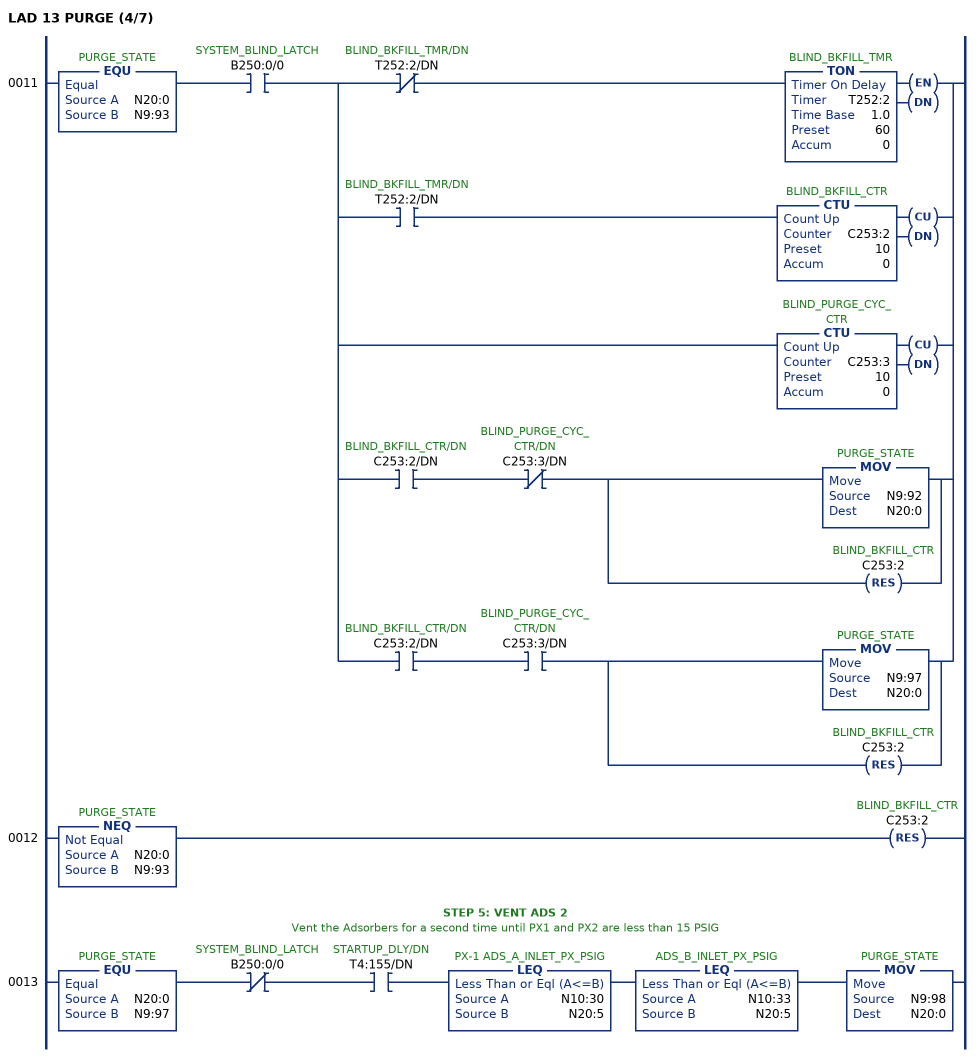
% Rung: 11 %
SOR EQU N20:0 N9:93 XIC B250:0/0 BST XIO T252:2/DN TON T252:2 1.0 60 0 NXB XIC T252:2/DN CTU C253:2 10 0 NXB CTU C253:3 10 0 NXB XIC C253:2/DN XIO C253:3/DN BST MOV N9:92 N20:0 NXB RES C253:2 BND NXB XIC C253:2/DN XIC C253:3/DN BST MOV N9:97 N20:0 NXB RES C253:2 BND BND EOR
%   N20:0  PURGE_STATE %
%   N9:93  PURGE_BACKFILL %
%   B250:0/0  SYSTEM_BLIND_LATCH %
%   T252:2  BLIND_BKFILL_TMR %
%   C253:2  BLIND_BKFILL_CTR %
%   C253:3  BLIND_PURGE_CYC_CTR %
%   N9:92  PURGE_VENT_ADSORBER %
%   N9:97  PURGE_VENT_ADS_2 %
% Rung: 12 %
SOR NEQ N20:0 N9:93 RES C253:2 EOR
%   N20:0  PURGE_STATE %
%   N9:93  PURGE_BACKFILL %
%   C253:2  BLIND_BKFILL_CTR %
% Rung: 13 %
% TITLE: STEP 5: VENT ADS 2 %
% Vent the Adsorbers for a second time until PX1 and PX2 are less than 15 PSIG %
SOR EQU N20:0 N9:97 XIO B250:0/0 XIC T4:155/DN LEQ N10:30 N20:5 LEQ N10:33 N20:5 MOV N9:98 N20:0 EOR
%   N20:0  PURGE_STATE %
%   N9:97  PURGE_VENT_ADS_2 %
%   B250:0/0  SYSTEM_BLIND_LATCH %
%   T4:155  STARTUP_DLY %
%   N10:30  ADS_A_INLET_PX_PSIG  "PX-1" %
%   N20:5  PURGE_VENT_ADS_2_PX %
%   N10:33  ADS_B_INLET_PX_PSIG %
%   N9:98  PURGE_VENT_GET_2 %

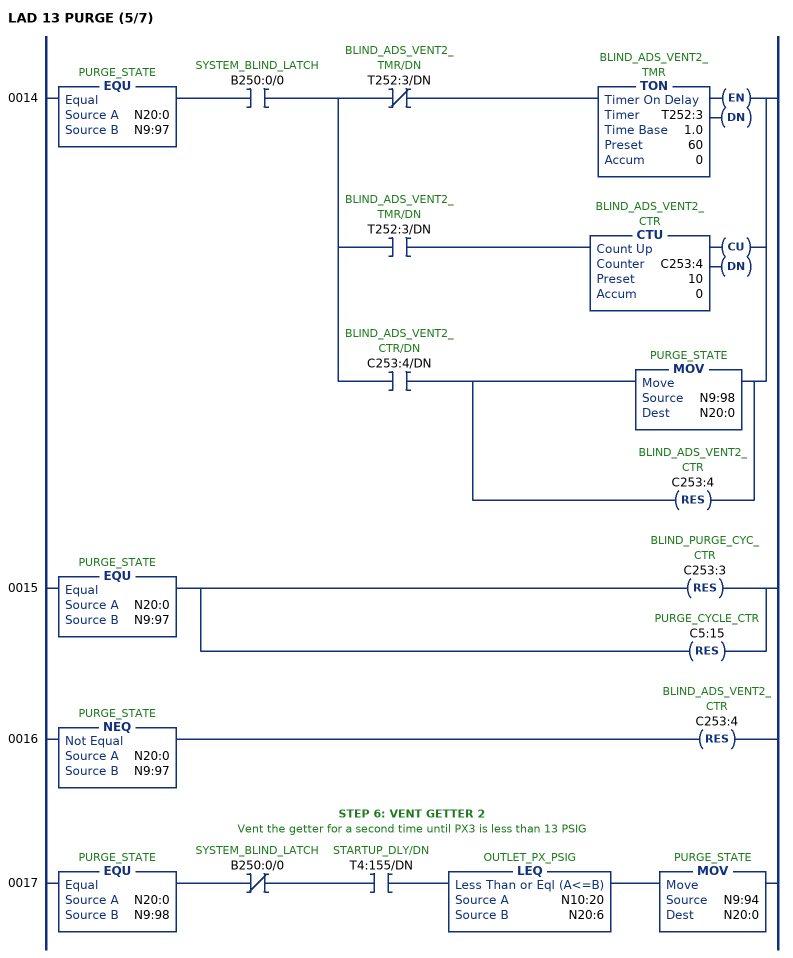
% Rung: 14 %
SOR EQU N20:0 N9:97 XIC B250:0/0 BST XIO T252:3/DN TON T252:3 1.0 60 0 NXB XIC T252:3/DN CTU C253:4 10 0 NXB XIC C253:4/DN BST MOV N9:98 N20:0 NXB RES C253:4 BND BND EOR
%   N20:0  PURGE_STATE %
%   N9:97  PURGE_VENT_ADS_2 %
%   B250:0/0  SYSTEM_BLIND_LATCH %
%   T252:3  BLIND_ADS_VENT2_TMR %
%   C253:4  BLIND_ADS_VENT2_CTR %
%   N9:98  PURGE_VENT_GET_2 %
% Rung: 15 %
SOR EQU N20:0 N9:97 BST RES C253:3 NXB RES C5:15 BND EOR
%   N20:0  PURGE_STATE %
%   N9:97  PURGE_VENT_ADS_2 %
%   C253:3  BLIND_PURGE_CYC_CTR %
%   C5:15  PURGE_CYCLE_CTR %
% Rung: 16 %
SOR NEQ N20:0 N9:97 RES C253:4 EOR
%   N20:0  PURGE_STATE %
%   N9:97  PURGE_VENT_ADS_2 %
%   C253:4  BLIND_ADS_VENT2_CTR %
% Rung: 17 %
% TITLE: STEP 6: VENT GETTER 2 %
% Vent the getter for a second time until PX3 is less than 13 PSIG %
SOR EQU N20:0 N9:98 XIO B250:0/0 XIC T4:155/DN LEQ N10:20 N20:6 MOV N9:94 N20:0 EOR
%   N20:0  PURGE_STATE %
%   N9:98  PURGE_VENT_GET_2 %
%   B250:0/0  SYSTEM_BLIND_LATCH %
%   T4:155  STARTUP_DLY %
%   N10:20  OUTLET_PX_PSIG %
%   N20:6  PURGE_VENT_GET_2_PX %
%   N9:94  PURGE_FINAL_VENT %

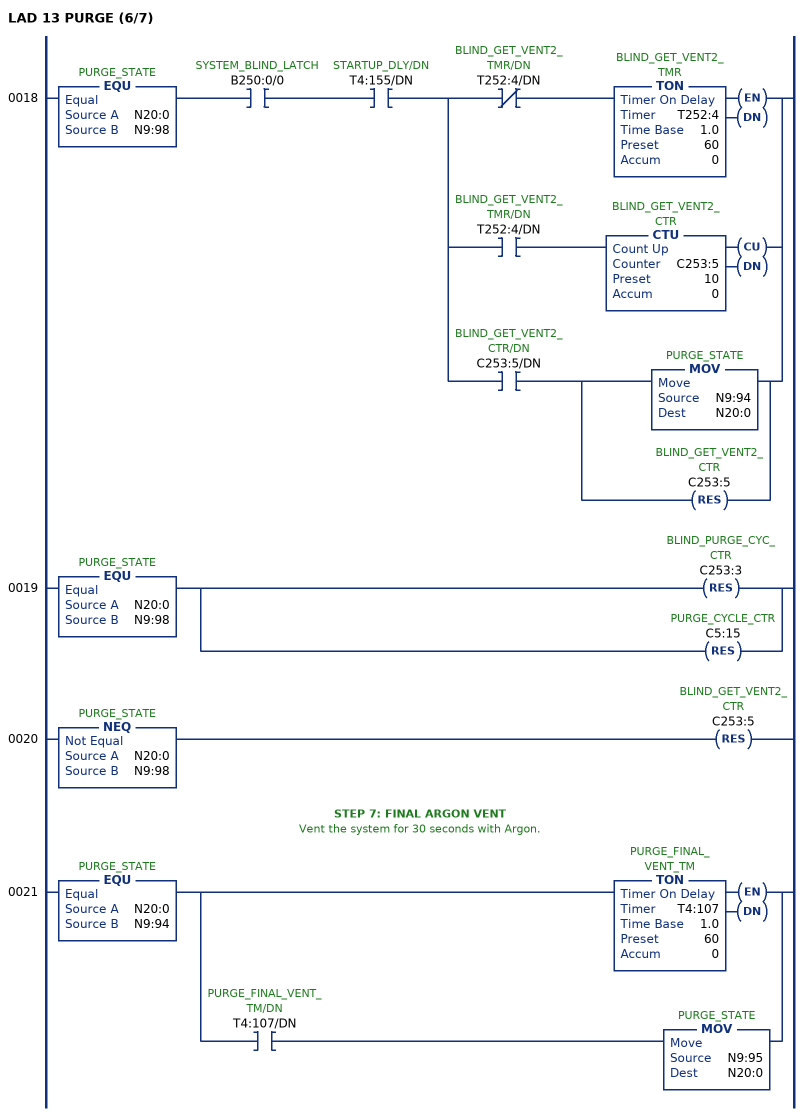
% Rung: 18 %
SOR EQU N20:0 N9:98 XIC B250:0/0 XIC T4:155/DN BST XIO T252:4/DN TON T252:4 1.0 60 0 NXB XIC T252:4/DN CTU C253:5 10 0 NXB XIC C253:5/DN BST MOV N9:94 N20:0 NXB RES C253:5 BND BND EOR
%   N20:0  PURGE_STATE %
%   N9:98  PURGE_VENT_GET_2 %
%   B250:0/0  SYSTEM_BLIND_LATCH %
%   T4:155  STARTUP_DLY %
%   T252:4  BLIND_GET_VENT2_TMR %
%   C253:5  BLIND_GET_VENT2_CTR %
%   N9:94  PURGE_FINAL_VENT %
% Rung: 19 %
SOR EQU N20:0 N9:98 BST RES C253:3 NXB RES C5:15 BND EOR
%   N20:0  PURGE_STATE %
%   N9:98  PURGE_VENT_GET_2 %
%   C253:3  BLIND_PURGE_CYC_CTR %
%   C5:15  PURGE_CYCLE_CTR %
% Rung: 20 %
SOR NEQ N20:0 N9:98 RES C253:5 EOR
%   N20:0  PURGE_STATE %
%   N9:98  PURGE_VENT_GET_2 %
%   C253:5  BLIND_GET_VENT2_CTR %
% Rung: 21 %
% TITLE: STEP 7: FINAL ARGON VENT %
% Vent the system for 30 seconds with Argon. %
SOR EQU N20:0 N9:94 BST TON T4:107 1.0 60 0 NXB XIC T4:107/DN MOV N9:95 N20:0 BND EOR
%   N20:0  PURGE_STATE %
%   N9:94  PURGE_FINAL_VENT %
%   T4:107  PURGE_FINAL_VENT_TM %
%   N9:95  PURGE_DONE %

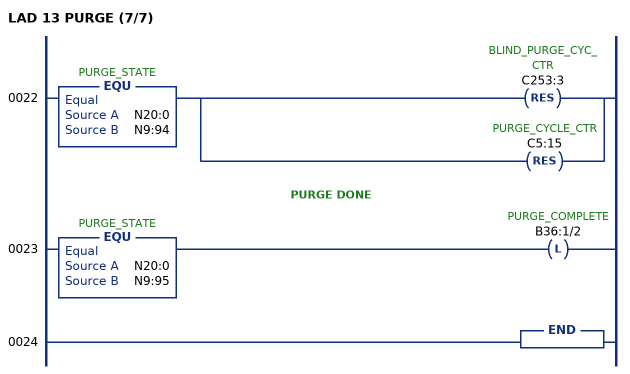
% Rung: 22 %
SOR EQU N20:0 N9:94 BST RES C253:3 NXB RES C5:15 BND EOR
%   N20:0  PURGE_STATE %
%   N9:94  PURGE_FINAL_VENT %
%   C253:3  BLIND_PURGE_CYC_CTR %
%   C5:15  PURGE_CYCLE_CTR %
% Rung: 23 %
% TITLE: PURGE DONE %
SOR EQU N20:0 N9:95 OTL B36:1/2 EOR
%   N20:0  PURGE_STATE %
%   N9:95  PURGE_DONE %
%   B36:1/2  PURGE_COMPLETE %
% Rung: 24 %
SOR END EOR

LADDER 14 "MFM"
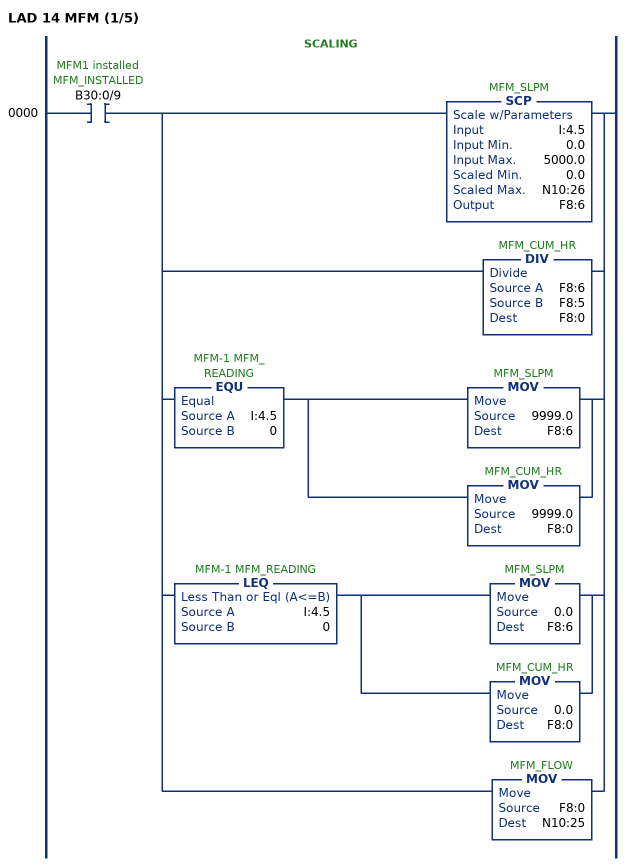
% Rung: 0 %
% TITLE: SCALING %
SOR XIC B30:0/9 BST SCP I:4.5 0.0 5000.0 0.0 N10:26 F8:6 NXB DIV F8:6 F8:5 F8:0 NXB EQU I:4.5 0 BST MOV 9999.0 F8:6 NXB MOV 9999.0 F8:0 BND NXB LEQ I:4.5 0 BST MOV 0.0 F8:6 NXB MOV 0.0 F8:0 BND NXB MOV F8:0 N10:25 BND EOR
%   B30:0/9  MFM_INSTALLED  "MFM1 installed" %
%   I:4.5  MFM_READING  "MFM-1" %
%   N10:26  MFM_SCALING %
%   F8:6  MFM_SLPM %
%   F8:5  CUM_TO_SLPM %
%   F8:0  MFM_CUM_HR %
%   N10:25  MFM_FLOW %

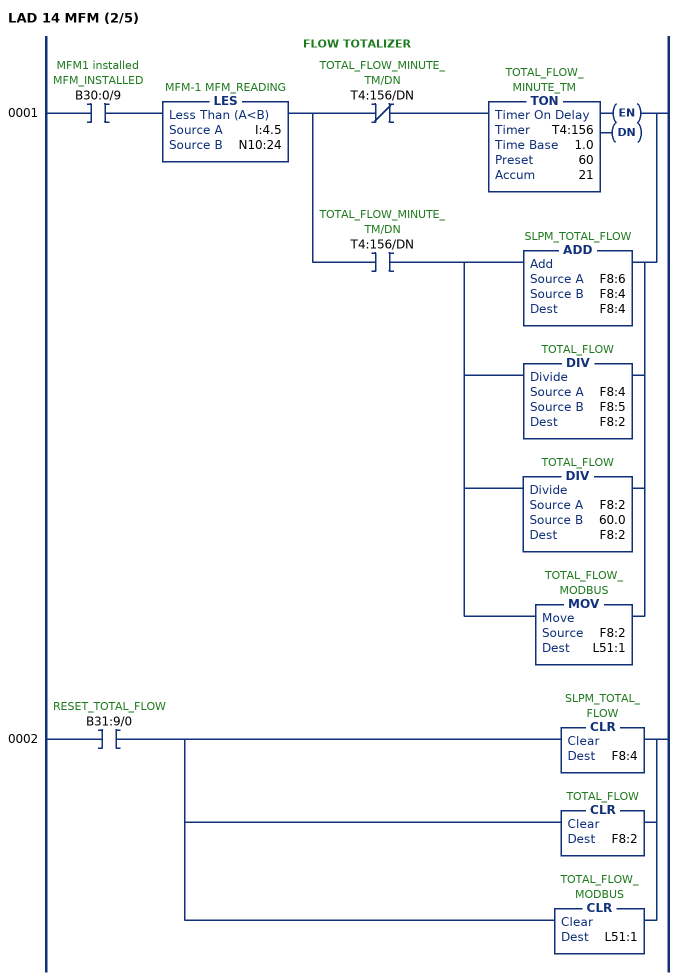
% Rung: 1 %
% TITLE: FLOW TOTALIZER %
SOR XIC B30:0/9 LES I:4.5 N10:24 BST XIO T4:156/DN TON T4:156 1.0 60 21 NXB XIC T4:156/DN BST ADD F8:6 F8:4 F8:4 NXB DIV F8:4 F8:5 F8:2 NXB DIV F8:2 60.0 F8:2 NXB MOV F8:2 L51:1 BND BND EOR
%   B30:0/9  MFM_INSTALLED  "MFM1 installed" %
%   I:4.5  MFM_READING  "MFM-1" %
%   N10:24  OPEN_MFM_5V %
%   T4:156  TOTAL_FLOW_MINUTE_TM %
%   F8:6  MFM_SLPM %
%   F8:4  SLPM_TOTAL_FLOW %
%   F8:5  CUM_TO_SLPM %
%   F8:2  TOTAL_FLOW %
%   L51:1  TOTAL_FLOW_MODBUS %
% Rung: 2 %
SOR XIC B31:9/0 BST CLR F8:4 NXB CLR F8:2 NXB CLR L51:1 BND EOR
%   B31:9/0  RESET_TOTAL_FLOW %
%   F8:4  SLPM_TOTAL_FLOW %
%   F8:2  TOTAL_FLOW %
%   L51:1  TOTAL_FLOW_MODBUS %

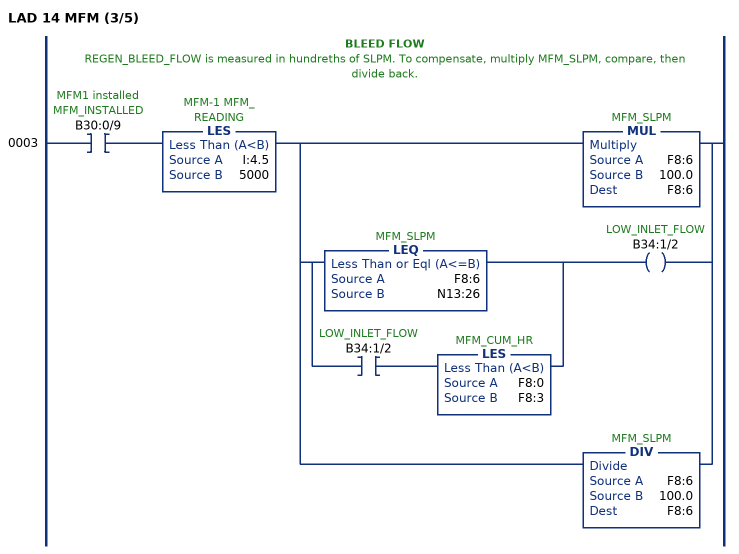
% Rung: 3 %
% TITLE: BLEED FLOW %
% REGEN_BLEED_FLOW is measured in hundreths of SLPM. To compensate, multiply MFM_SLPM, compare, then divide back. %
SOR XIC B30:0/9 LES I:4.5 5000 BST MUL F8:6 100.0 F8:6 NXB BST LEQ F8:6 N13:26 NXB XIC B34:1/2 LES F8:0 F8:3 BND OTE B34:1/2 NXB DIV F8:6 100.0 F8:6 BND EOR
%   B30:0/9  MFM_INSTALLED  "MFM1 installed" %
%   I:4.5  MFM_READING  "MFM-1" %
%   F8:6  MFM_SLPM %
%   N13:26  REGEN_BLEED_FLOW %
%   B34:1/2  LOW_INLET_FLOW %
%   F8:0  MFM_CUM_HR %
%   F8:3  BLEED_FLOW_CUTOFF %

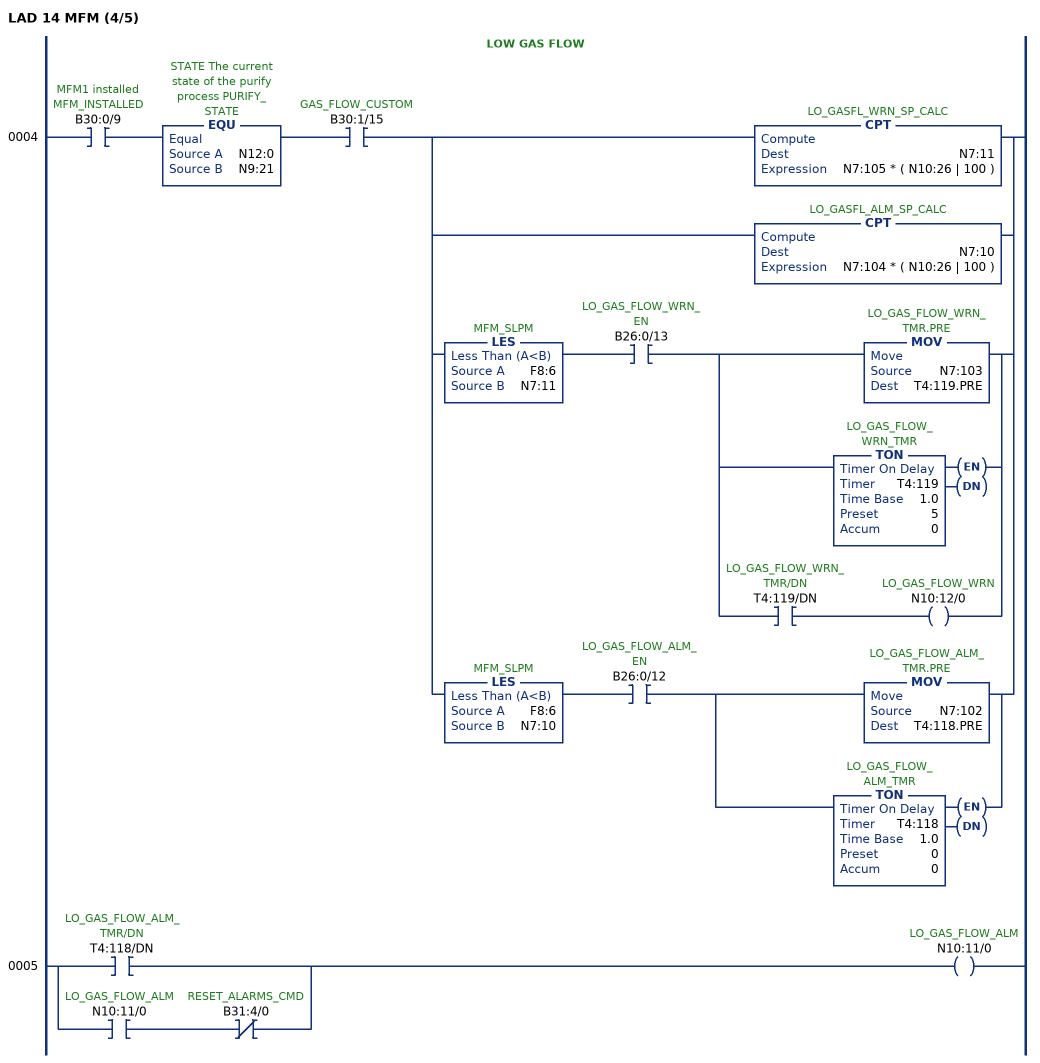
% Rung: 4 %
% TITLE: LOW GAS FLOW %
SOR XIC B30:0/9 EQU N12:0 N9:21 XIC B30:1/15 BST CPT N7:11 " N7:105 * ( N10:26 | 100 ) " NXB CPT N7:10 " N7:104 * ( N10:26 | 100 ) " NXB LES F8:6 N7:11 XIC B26:0/13 BST MOV N7:103 T4:119.PRE NXB TON T4:119 1.0 5 0 NXB XIC T4:119/DN OTE N10:12/0 BND NXB LES F8:6 N7:10 XIC B26:0/12 BST MOV N7:102 T4:118.PRE NXB TON T4:118 1.0 0 0 BND BND EOR
%   B30:0/9  MFM_INSTALLED  "MFM1 installed" %
%   N12:0  PURIFY_STATE  "STATE The current state of the purify process" %
%   N9:21  PURIFY_RUN  "STATE Purify running" %
%   B30:1/15  GAS_FLOW_CUSTOM %
%   N7:11  LO_GASFL_WRN_SP_CALC %
%   N7:105  LO_GAS_FLOW_WRN_SP %
%   N10:26  MFM_SCALING %
%   N7:10  LO_GASFL_ALM_SP_CALC %
%   N7:104  LO_GAS_FLOW_ALM_SP %
%   F8:6  MFM_SLPM %
%   B26:0/13  LO_GAS_FLOW_WRN_EN %
%   N7:103  LO_GAS_FLOW_WRN_DLY %
%   T4:119  LO_GAS_FLOW_WRN_TMR %
%   N10:12/0  LO_GAS_FLOW_WRN %
%   B26:0/12  LO_GAS_FLOW_ALM_EN %
%   N7:102  LO_GAS_FLOW_ALM_DLY %
%   T4:118  LO_GAS_FLOW_ALM_TMR %
% Rung: 5 %
SOR BST XIC T4:118/DN NXB XIC N10:11/0 XIO B31:4/0 BND OTE N10:11/0 EOR
%   T4:118  LO_GAS_FLOW_ALM_TMR %
%   N10:11/0  LO_GAS_FLOW_ALM %
%   B31:4/0  RESET_ALARMS_CMD %

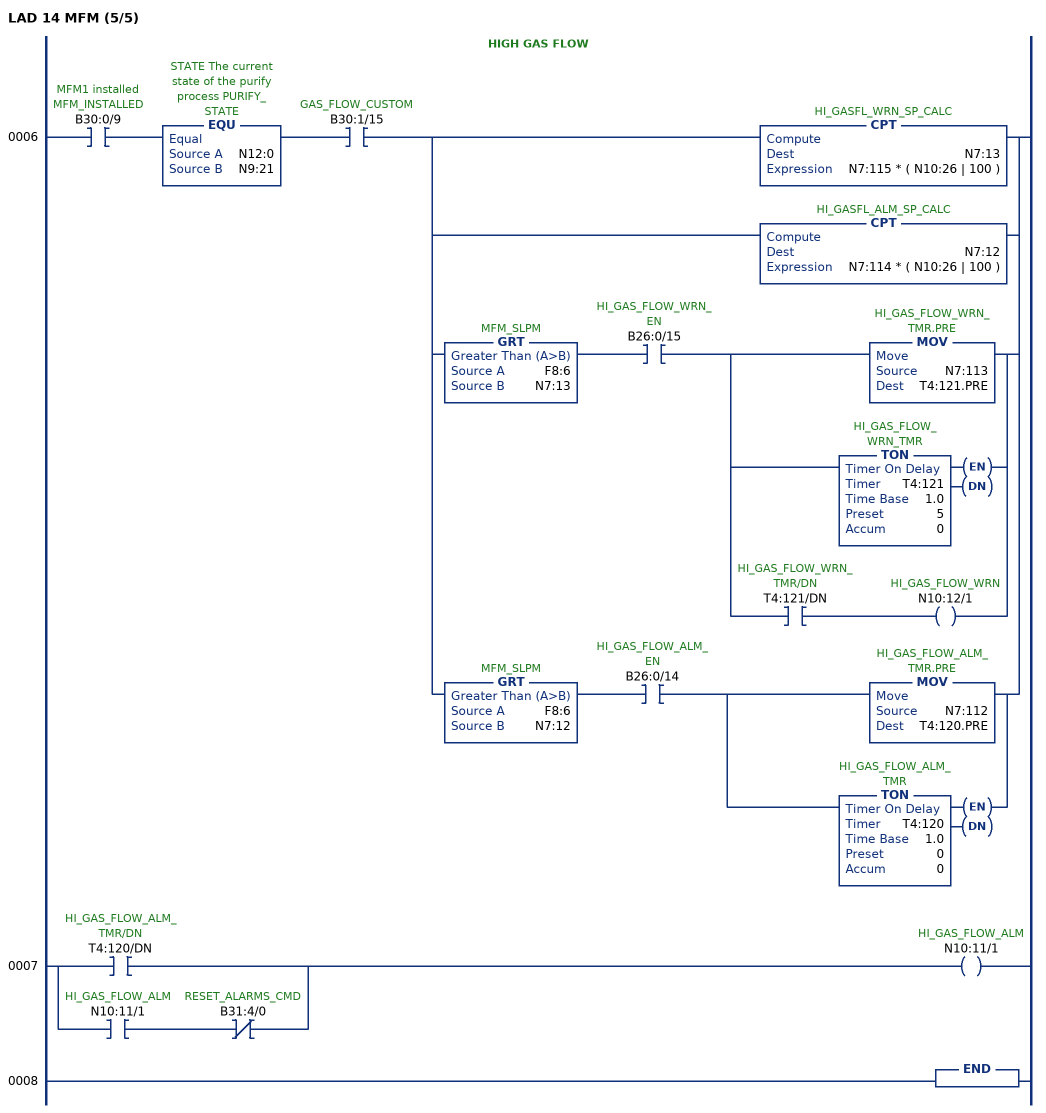
% Rung: 6 %
% TITLE: HIGH GAS FLOW %
SOR XIC B30:0/9 EQU N12:0 N9:21 XIC B30:1/15 BST CPT N7:13 " N7:115 * ( N10:26 | 100 ) " NXB CPT N7:12 " N7:114 * ( N10:26 | 100 ) " NXB GRT F8:6 N7:13 XIC B26:0/15 BST MOV N7:113 T4:121.PRE NXB TON T4:121 1.0 5 0 NXB XIC T4:121/DN OTE N10:12/1 BND NXB GRT F8:6 N7:12 XIC B26:0/14 BST MOV N7:112 T4:120.PRE NXB TON T4:120 1.0 0 0 BND BND EOR
%   B30:0/9  MFM_INSTALLED  "MFM1 installed" %
%   N12:0  PURIFY_STATE  "STATE The current state of the purify process" %
%   N9:21  PURIFY_RUN  "STATE Purify running" %
%   B30:1/15  GAS_FLOW_CUSTOM %
%   N7:13  HI_GASFL_WRN_SP_CALC %
%   N7:115  HI_GAS_FLOW_WRN_SP %
%   N10:26  MFM_SCALING %
%   N7:12  HI_GASFL_ALM_SP_CALC %
%   N7:114  HI_GAS_FLOW_ALM_SP %
%   F8:6  MFM_SLPM %
%   B26:0/15  HI_GAS_FLOW_WRN_EN %
%   N7:113  HI_GAS_FLOW_WRN_DLY %
%   T4:121  HI_GAS_FLOW_WRN_TMR %
%   N10:12/1  HI_GAS_FLOW_WRN %
%   B26:0/14  HI_GAS_FLOW_ALM_EN %
%   N7:112  HI_GAS_FLOW_ALM_DLY %
%   T4:120  HI_GAS_FLOW_ALM_TMR %
% Rung: 7 %
SOR BST XIC T4:120/DN NXB XIC N10:11/1 XIO B31:4/0 BND OTE N10:11/1 EOR
%   T4:120  HI_GAS_FLOW_ALM_TMR %
%   N10:11/1  HI_GAS_FLOW_ALM %
%   B31:4/0  RESET_ALARMS_CMD %
% Rung: 8 %
SOR END EOR

LADDER 16 "MFC"
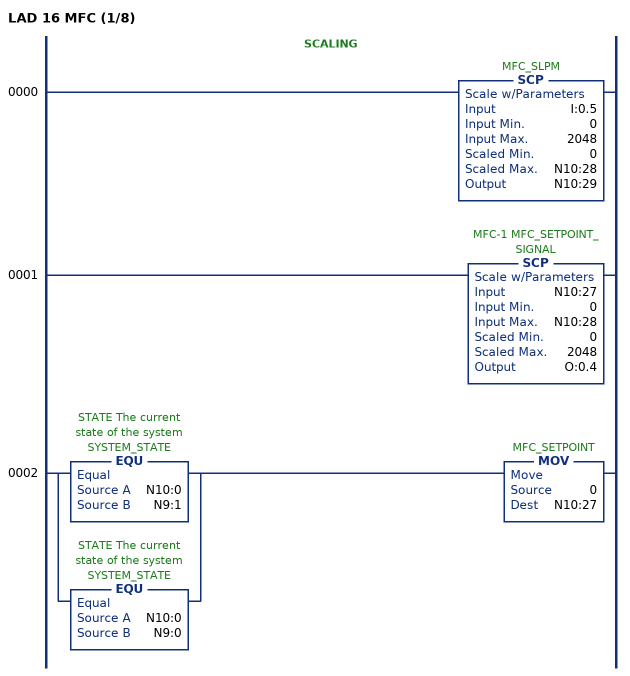
% Rung: 0 %
% TITLE: SCALING %
SOR SCP I:0.5 0 2048 0 N10:28 N10:29 EOR
%   I:0.5  MFC_FEEDBACK  "MFC-1" %
%   N10:28  MFC_SCALING  "in slpm" %
%   N10:29  MFC_SLPM %
% Rung: 1 %
SOR SCP N10:27 0 N10:28 0 2048 O:0.4 EOR
%   N10:27  MFC_SETPOINT %
%   N10:28  MFC_SCALING  "in slpm" %
%   O:0.4  MFC_SETPOINT_SIGNAL  "MFC-1" %
% Rung: 2 %
SOR BST EQU N10:0 N9:1 NXB EQU N10:0 N9:0 BND MOV 0 N10:27 EOR
%   N10:0  SYSTEM_STATE  "STATE The current state of the system" %
%   N9:1  SYSTEM_STANDBY  "STATE System Process" %
%   N9:0  SYSTEM_OFFLINE %
%   N10:27  MFC_SETPOINT %

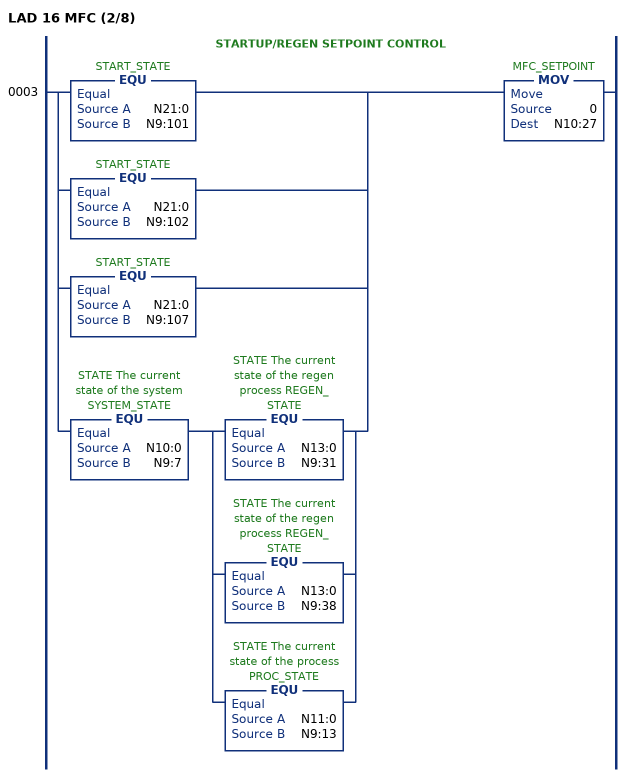
% Rung: 3 %
% TITLE: STARTUP/REGEN SETPOINT CONTROL %
SOR BST EQU N21:0 N9:101 NXB EQU N21:0 N9:102 NXB EQU N21:0 N9:107 NXB EQU N10:0 N9:7 BST EQU N13:0 N9:31 NXB EQU N13:0 N9:38 NXB EQU N11:0 N9:13 BND BND MOV 0 N10:27 EOR
%   N21:0  START_STATE %
%   N9:101  START_COOL %
%   N9:102  START_VENT_ADS_1 %
%   N9:107  START_VENT_ADS_2 %
%   N10:0  SYSTEM_STATE  "STATE The current state of the system" %
%   N9:7  SYSTEM_COLD_START %
%   N13:0  REGEN_STATE  "STATE The current state of the regen process" %
%   N9:31  REGEN_DELAY  "STATE Regen Delay" %
%   N9:38  REGEN_DONE %
%   N11:0  PROC_STATE  "STATE The current state of the process" %
%   N9:13  PROC_OVERLAP  "STATE Process Purify Overlap" %
%   N10:27  MFC_SETPOINT %

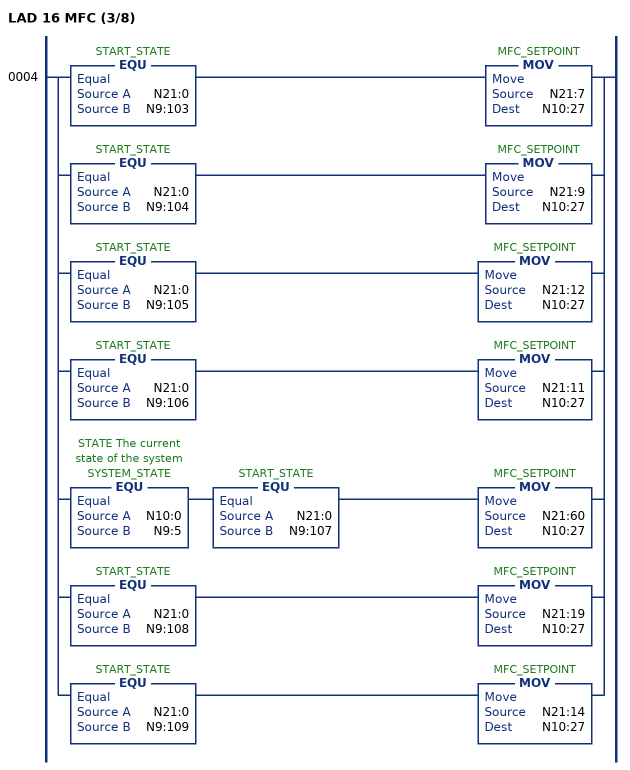
% Rung: 4 %
SOR BST EQU N21:0 N9:103 MOV N21:7 N10:27 NXB EQU N21:0 N9:104 MOV N21:9 N10:27 NXB EQU N21:0 N9:105 MOV N21:12 N10:27 NXB EQU N21:0 N9:106 MOV N21:11 N10:27 NXB EQU N10:0 N9:5 EQU N21:0 N9:107 MOV N21:60 N10:27 NXB EQU N21:0 N9:108 MOV N21:19 N10:27 NXB EQU N21:0 N9:109 MOV N21:14 N10:27 BND EOR
%   N21:0  START_STATE %
%   N9:103  START_VENT_GET_1 %
%   N21:7  START_VENT_GET_1_FLW %
%   N10:27  MFC_SETPOINT %
%   N9:104  START_HEAT_GETTER %
%   N21:9  START_HEAT_FLW %
%   N9:105  START_VENT_ALL %
%   N21:12  START_VENT_ALL_FLW %
%   N9:106  START_BACKFILL_1 %
%   N21:11  START_BKFIL_1_FLW %
%   N10:0  SYSTEM_STATE  "STATE The current state of the system" %
%   N9:5  SYSTEM_QUICK_START %
%   N9:107  START_VENT_ADS_2 %
%   N21:60  START_VENT_ADS_2_FLW %
%   N9:108  START_VENT_GET_2 %
%   N21:19  START_VENT_GET_2_FLW %
%   N9:109  START_BKFL_2 %
%   N21:14  START_BKFIL_2_FLW %

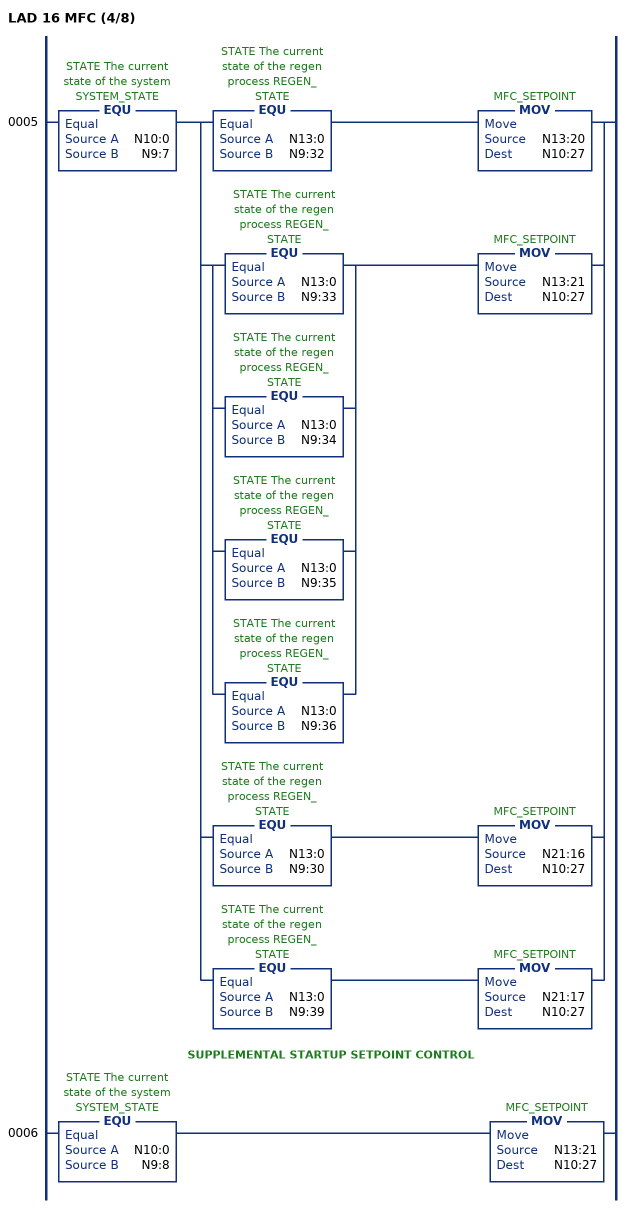
% Rung: 5 %
SOR EQU N10:0 N9:7 BST EQU N13:0 N9:32 MOV N13:20 N10:27 NXB BST EQU N13:0 N9:33 NXB EQU N13:0 N9:34 NXB EQU N13:0 N9:35 NXB EQU N13:0 N9:36 BND MOV N13:21 N10:27 NXB EQU N13:0 N9:30 MOV N21:16 N10:27 NXB EQU N13:0 N9:39 MOV N21:17 N10:27 BND EOR
%   N10:0  SYSTEM_STATE  "STATE The current state of the system" %
%   N9:7  SYSTEM_COLD_START %
%   N13:0  REGEN_STATE  "STATE The current state of the regen process" %
%   N9:32  REGEN_VENT  "STATE Regen Vent" %
%   N13:20  REGEN_VENT_FLOW %
%   N10:27  MFC_SETPOINT %
%   N9:33  REGEN_HEAT_BED  "STATE Regen Heat wall" %
%   N9:34  REGEN_RUN  "STATE Regen Running" %
%   N9:35  REGEN_COOL_WALL  "STATE Regen Cool wall" %
%   N9:36  REGEN_COOL  "STATE Regen Cool" %
%   N13:21  REGEN_MAIN_FLOW %
%   N9:30  REGEN_STANDBY  "STATE Regen Standby" %
%   N21:16  START_REG_BLEED_FLW %
%   N9:39  REGEN_BACKFILL %
%   N21:17  START_REG_BKFIL_FLW %
% Rung: 6 %
% TITLE: SUPPLEMENTAL STARTUP SETPOINT CONTROL %
SOR EQU N10:0 N9:8 MOV N13:21 N10:27 EOR
%   N10:0  SYSTEM_STATE  "STATE The current state of the system" %
%   N9:8  SYSTEM_SUPPLEMENTAL %
%   N13:21  REGEN_MAIN_FLOW %
%   N10:27  MFC_SETPOINT %

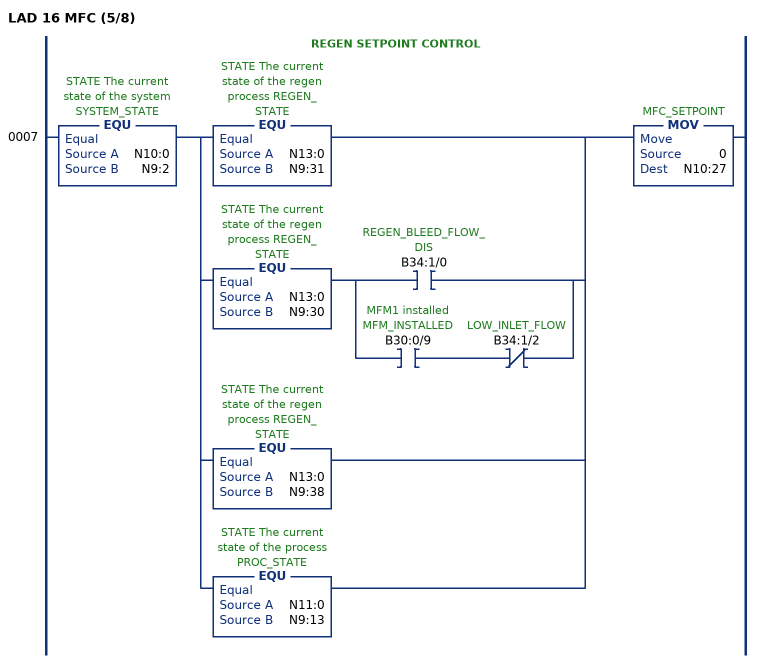
% Rung: 7 %
% TITLE: REGEN SETPOINT CONTROL %
SOR EQU N10:0 N9:2 BST EQU N13:0 N9:31 NXB EQU N13:0 N9:30 BST XIC B34:1/0 NXB XIC B30:0/9 XIO B34:1/2 BND NXB EQU N13:0 N9:38 NXB EQU N11:0 N9:13 BND MOV 0 N10:27 EOR
%   N10:0  SYSTEM_STATE  "STATE The current state of the system" %
%   N9:2  SYSTEM_PROCESS  "STATE System Process" %
%   N13:0  REGEN_STATE  "STATE The current state of the regen process" %
%   N9:31  REGEN_DELAY  "STATE Regen Delay" %
%   N9:30  REGEN_STANDBY  "STATE Regen Standby" %
%   B34:1/0  REGEN_BLEED_FLOW_DIS %
%   B30:0/9  MFM_INSTALLED  "MFM1 installed" %
%   B34:1/2  LOW_INLET_FLOW %
%   N9:38  REGEN_DONE %
%   N11:0  PROC_STATE  "STATE The current state of the process" %
%   N9:13  PROC_OVERLAP  "STATE Process Purify Overlap" %
%   N10:27  MFC_SETPOINT %

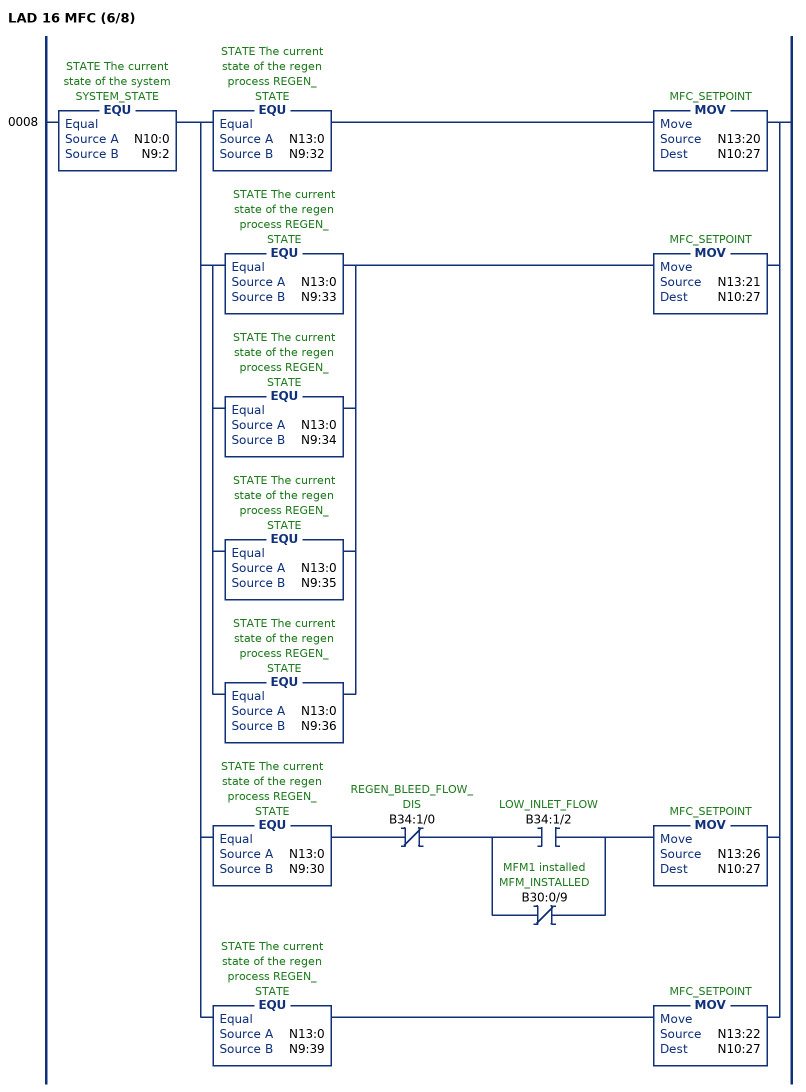
% Rung: 8 %
SOR EQU N10:0 N9:2 BST EQU N13:0 N9:32 MOV N13:20 N10:27 NXB BST EQU N13:0 N9:33 NXB EQU N13:0 N9:34 NXB EQU N13:0 N9:35 NXB EQU N13:0 N9:36 BND MOV N13:21 N10:27 NXB EQU N13:0 N9:30 XIO B34:1/0 BST XIC B34:1/2 NXB XIO B30:0/9 BND MOV N13:26 N10:27 NXB EQU N13:0 N9:39 MOV N13:22 N10:27 BND EOR
%   N10:0  SYSTEM_STATE  "STATE The current state of the system" %
%   N9:2  SYSTEM_PROCESS  "STATE System Process" %
%   N13:0  REGEN_STATE  "STATE The current state of the regen process" %
%   N9:32  REGEN_VENT  "STATE Regen Vent" %
%   N13:20  REGEN_VENT_FLOW %
%   N10:27  MFC_SETPOINT %
%   N9:33  REGEN_HEAT_BED  "STATE Regen Heat wall" %
%   N9:34  REGEN_RUN  "STATE Regen Running" %
%   N9:35  REGEN_COOL_WALL  "STATE Regen Cool wall" %
%   N9:36  REGEN_COOL  "STATE Regen Cool" %
%   N13:21  REGEN_MAIN_FLOW %
%   N9:30  REGEN_STANDBY  "STATE Regen Standby" %
%   B34:1/0  REGEN_BLEED_FLOW_DIS %
%   B34:1/2  LOW_INLET_FLOW %
%   B30:0/9  MFM_INSTALLED  "MFM1 installed" %
%   N13:26  REGEN_BLEED_FLOW %
%   N9:39  REGEN_BACKFILL %
%   N13:22  REGEN_BACKFILL_FLOW %

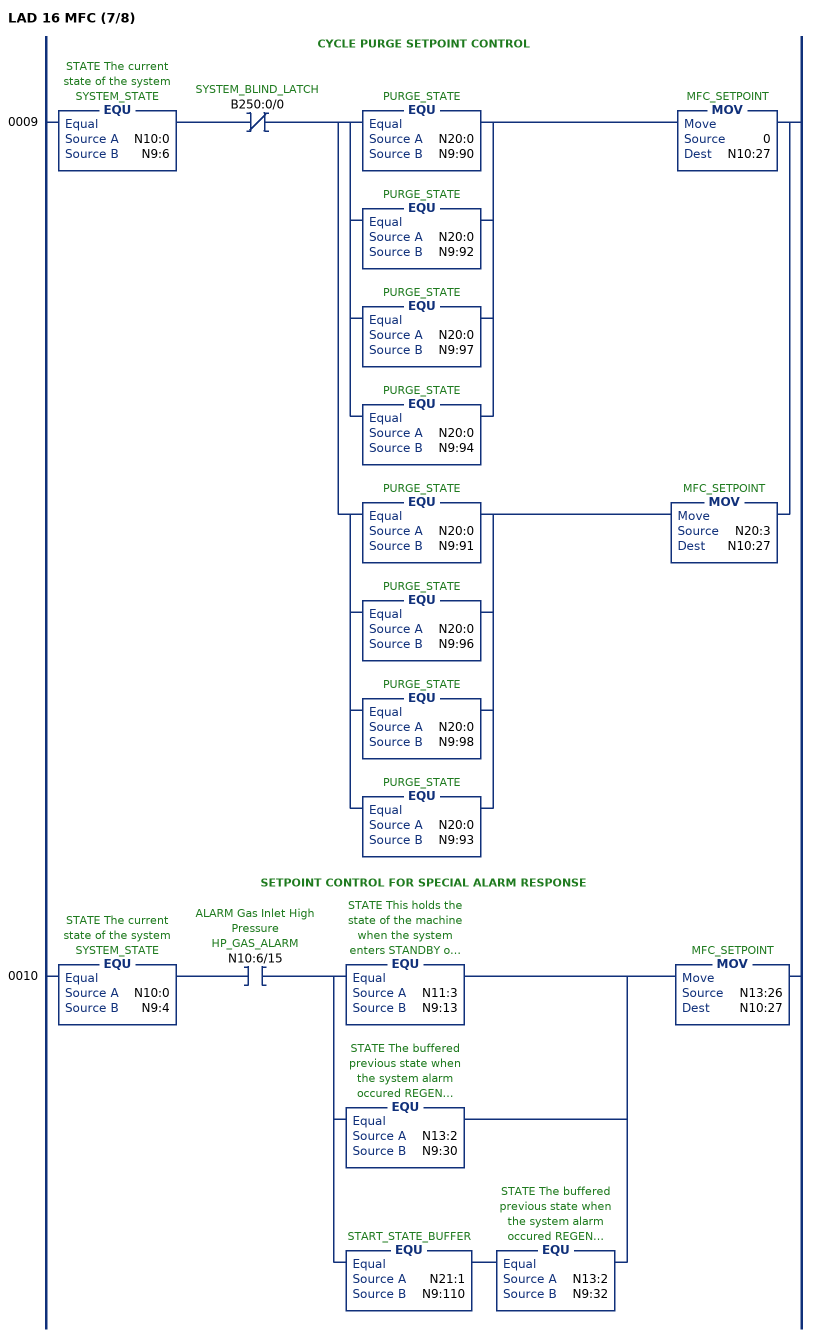
% Rung: 9 %
% TITLE: CYCLE PURGE SETPOINT CONTROL %
SOR EQU N10:0 N9:6 XIO B250:0/0 BST BST EQU N20:0 N9:90 NXB EQU N20:0 N9:92 NXB EQU N20:0 N9:97 NXB EQU N20:0 N9:94 BND MOV 0 N10:27 NXB BST EQU N20:0 N9:91 NXB EQU N20:0 N9:96 NXB EQU N20:0 N9:98 NXB EQU N20:0 N9:93 BND MOV N20:3 N10:27 BND EOR
%   N10:0  SYSTEM_STATE  "STATE The current state of the system" %
%   N9:6  SYSTEM_PURGE %
%   B250:0/0  SYSTEM_BLIND_LATCH %
%   N20:0  PURGE_STATE %
%   N9:90  PURGE_IDLE %
%   N9:92  PURGE_VENT_ADSORBER %
%   N9:97  PURGE_VENT_ADS_2 %
%   N9:94  PURGE_FINAL_VENT %
%   N10:27  MFC_SETPOINT %
%   N9:91  PURGE_INIT_VENT %
%   N9:96  PURGE_VENT_GETTER %
%   N9:98  PURGE_VENT_GET_2 %
%   N9:93  PURGE_BACKFILL %
%   N20:3  PURGE_FLOW %
% Rung: 10 %
% TITLE: SETPOINT CONTROL FOR SPECIAL ALARM RESPONSE %
SOR EQU N10:0 N9:4 XIC N10:6/15 BST EQU N11:3 N9:13 NXB EQU N13:2 N9:30 NXB EQU N21:1 N9:110 EQU N13:2 N9:32 BND MOV N13:26 N10:27 EOR
%   N10:0  SYSTEM_STATE  "STATE The current state of the system" %
%   N9:4  SYSTEM_ALARM  "STATE System Alarm" %
%   N10:6/15  HP_GAS_ALARM  "ALARM Gas Inlet High Pressure" %
%   N11:3  PROC_STATE_BUFFER  "STATE This holds the state of the machine when the system enters STANDBY or ALARM" %
%   N9:13  PROC_OVERLAP  "STATE Process Purify Overlap" %
%   N13:2  REGEN_SYSTEM_BUFFER  "STATE The buffered previous state when the system alarm occured" %
%   N9:30  REGEN_STANDBY  "STATE Regen Standby" %
%   N21:1  START_STATE_BUFFER %
%   N9:110  START_REG_VENT %
%   N9:32  REGEN_VENT  "STATE Regen Vent" %
%   N13:26  REGEN_BLEED_FLOW %
%   N10:27  MFC_SETPOINT %

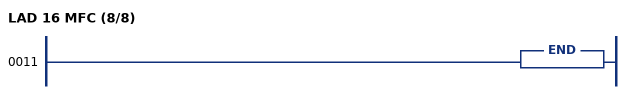
% Rung: 11 %
SOR END EOR

LADDER 17 "BYPASS"    % Controls the bypass %
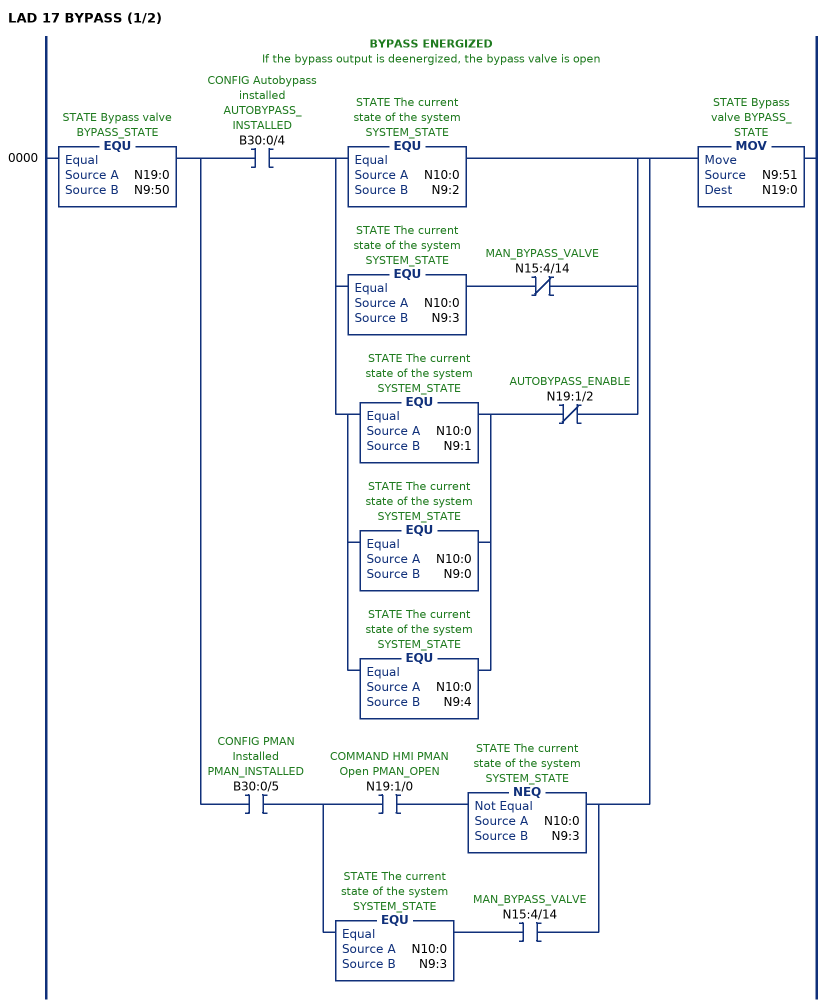
% Rung: 0 %
% TITLE: BYPASS ENERGIZED %
% If the bypass output is deenergized, the bypass valve is open %
SOR EQU N19:0 N9:50 BST XIC B30:0/4 BST EQU N10:0 N9:2 NXB EQU N10:0 N9:3 XIO N15:4/14 NXB BST EQU N10:0 N9:1 NXB EQU N10:0 N9:0 NXB EQU N10:0 N9:4 BND XIO N19:1/2 BND NXB XIC B30:0/5 BST XIC N19:1/0 NEQ N10:0 N9:3 NXB EQU N10:0 N9:3 XIC N15:4/14 BND BND MOV N9:51 N19:0 EOR
%   N19:0  BYPASS_STATE  "STATE Bypass valve" %
%   N9:50  BYPASS_DEENERGIZED  "STATE Bypass Deenergized" %
%   B30:0/4  AUTOBYPASS_INSTALLED  "CONFIG Autobypass installed" %
%   N10:0  SYSTEM_STATE  "STATE The current state of the system" %
%   N9:2  SYSTEM_PROCESS  "STATE System Process" %
%   N9:3  SYSTEM_MANUAL  "STATE System Manual" %
%   N15:4/14  MAN_BYPASS_VALVE %
%   N9:1  SYSTEM_STANDBY  "STATE System Process" %
%   N9:0  SYSTEM_OFFLINE %
%   N9:4  SYSTEM_ALARM  "STATE System Alarm" %
%   N19:1/2  AUTOBYPASS_ENABLE %
%   B30:0/5  PMAN_INSTALLED  "CONFIG PMAN Installed" %
%   N19:1/0  PMAN_OPEN  "COMMAND HMI PMAN Open" %
%   N9:51  BYPASS_ENERGIZED  "STATE Bypass Energized" %

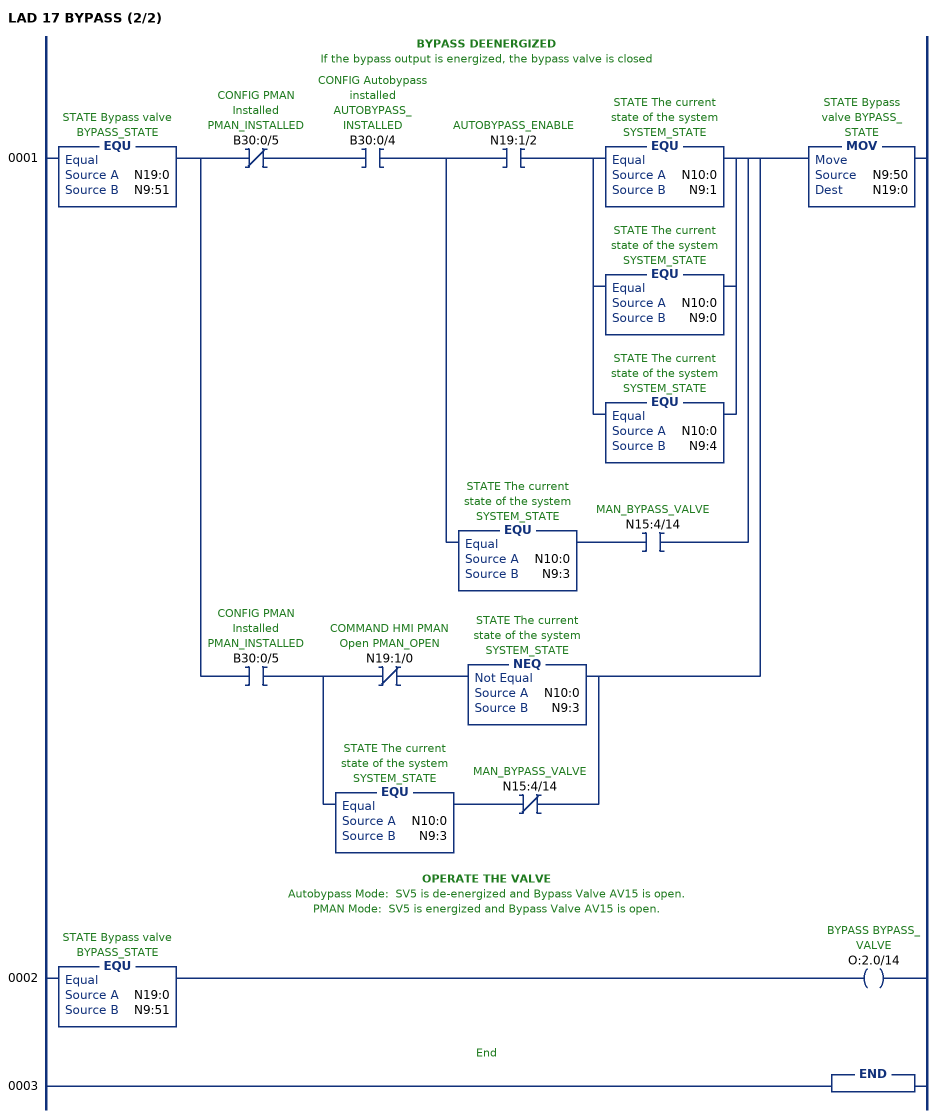
% Rung: 1 %
% TITLE: BYPASS DEENERGIZED %
% If the bypass output is energized, the bypass valve is closed %
SOR EQU N19:0 N9:51 BST XIO B30:0/5 XIC B30:0/4 BST XIC N19:1/2 BST EQU N10:0 N9:1 NXB EQU N10:0 N9:0 NXB EQU N10:0 N9:4 BND NXB EQU N10:0 N9:3 XIC N15:4/14 BND NXB XIC B30:0/5 BST XIO N19:1/0 NEQ N10:0 N9:3 NXB EQU N10:0 N9:3 XIO N15:4/14 BND BND MOV N9:50 N19:0 EOR
%   N19:0  BYPASS_STATE  "STATE Bypass valve" %
%   N9:51  BYPASS_ENERGIZED  "STATE Bypass Energized" %
%   B30:0/5  PMAN_INSTALLED  "CONFIG PMAN Installed" %
%   B30:0/4  AUTOBYPASS_INSTALLED  "CONFIG Autobypass installed" %
%   N19:1/2  AUTOBYPASS_ENABLE %
%   N10:0  SYSTEM_STATE  "STATE The current state of the system" %
%   N9:1  SYSTEM_STANDBY  "STATE System Process" %
%   N9:0  SYSTEM_OFFLINE %
%   N9:4  SYSTEM_ALARM  "STATE System Alarm" %
%   N9:3  SYSTEM_MANUAL  "STATE System Manual" %
%   N15:4/14  MAN_BYPASS_VALVE %
%   N19:1/0  PMAN_OPEN  "COMMAND HMI PMAN Open" %
%   N9:50  BYPASS_DEENERGIZED  "STATE Bypass Deenergized" %
% Rung: 2 %
% TITLE: OPERATE THE VALVE %
% Autobypass Mode:  SV5 is de-energized and Bypass Valve AV15 is open.
% PMAN Mode:  SV5 is energized and Bypass Valve AV15 is open. %
SOR EQU N19:0 N9:51 OTE O:2.0/14 EOR
%   N19:0  BYPASS_STATE  "STATE Bypass valve" %
%   N9:51  BYPASS_ENERGIZED  "STATE Bypass Energized" %
%   O:2.0/14  BYPASS_VALVE  "BYPASS" %
% Rung: 3 %
% End %
SOR END EOR

LADDER 20 "ADS A"    % Controls the Adsorber A %
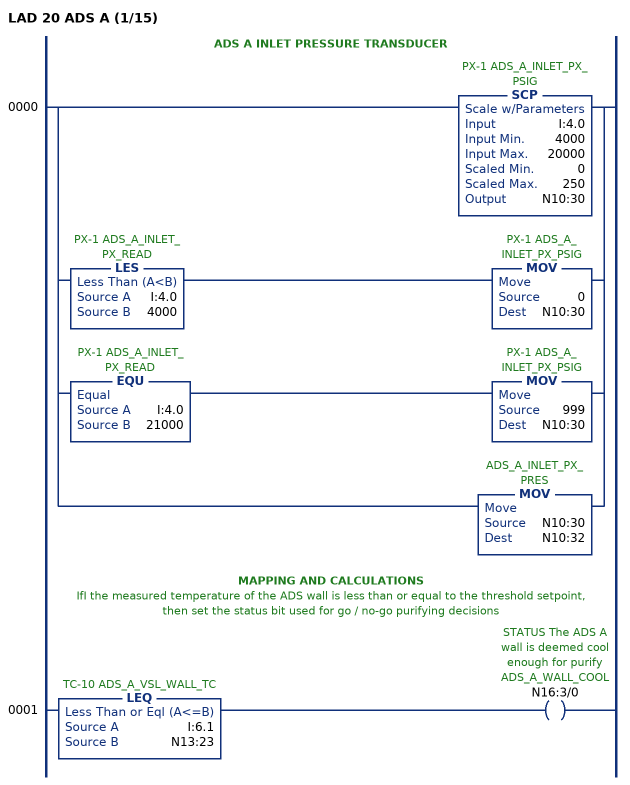
% Rung: 0 %
% TITLE: ADS A INLET PRESSURE TRANSDUCER %
SOR BST SCP I:4.0 4000 20000 0 250 N10:30 NXB LES I:4.0 4000 MOV 0 N10:30 NXB EQU I:4.0 21000 MOV 999 N10:30 NXB MOV N10:30 N10:32 BND EOR
%   I:4.0  ADS_A_INLET_PX_READ  "PX-1" %
%   N10:30  ADS_A_INLET_PX_PSIG  "PX-1" %
%   N10:32  ADS_A_INLET_PX_PRES %
% Rung: 1 %
% TITLE: MAPPING AND CALCULATIONS %
% IfI the measured temperature of the ADS wall is less than or equal to the threshold setpoint, then set the status bit used for go / no-go purifying decisions %
SOR LEQ I:6.1 N13:23 OTE N16:3/0 EOR
%   I:6.1  ADS_A_VSL_WALL_TC  "TC-10" %
%   N13:23  ADS_WALL_TEMP_COOL  "CONFIG The temp at which the adsorber wall is deemed to be cool enough to purify" %
%   N16:3/0  ADS_A_WALL_COOL  "STATUS The ADS A wall is deemed cool enough for purify" %

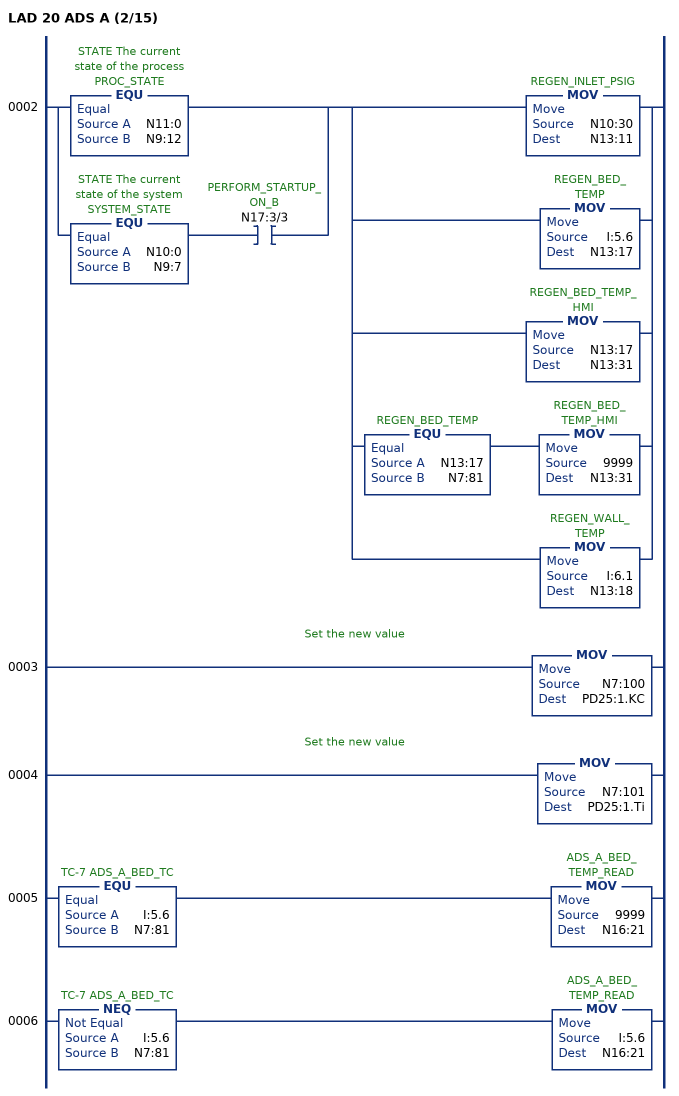
% Rung: 2 %
SOR BST EQU N11:0 N9:12 NXB EQU N10:0 N9:7 XIC N17:3/3 BND BST MOV N10:30 N13:11 NXB BST MOV I:5.6 N13:17 NXB MOV N13:17 N13:31 BND NXB EQU N13:17 N7:81 MOV 9999 N13:31 NXB MOV I:6.1 N13:18 BND EOR
%   N11:0  PROC_STATE  "STATE The current state of the process" %
%   N9:12  PROC_PFY_B_REG_A  "STATE Process Purify B" %
%   N10:0  SYSTEM_STATE  "STATE The current state of the system" %
%   N9:7  SYSTEM_COLD_START %
%   N17:3/3  PERFORM_STARTUP_ON_B %
%   N10:30  ADS_A_INLET_PX_PSIG  "PX-1" %
%   N13:11  REGEN_INLET_PSIG %
%   I:5.6  ADS_A_BED_TC  "TC-7" %
%   N13:17  REGEN_BED_TEMP %
%   N13:31  REGEN_BED_TEMP_HMI %
%   N7:81  TC_OPEN_SP  "CONFIG The value read by an open TC input" %
%   I:6.1  ADS_A_VSL_WALL_TC  "TC-10" %
%   N13:18  REGEN_WALL_TEMP %
% Rung: 3 %
% Set the new value %
SOR MOV N7:100 PD25:1.KC EOR
%   N7:100  BLANKET_P  "CONFIG Blanket Proportional Gain New" %
% Rung: 4 %
% Set the new value %
SOR MOV N7:101 PD25:1.Ti EOR
%   N7:101  BLANKET_I  "CONFIG Blanket Integral Gain New" %
% Rung: 5 %
SOR EQU I:5.6 N7:81 MOV 9999 N16:21 EOR
%   I:5.6  ADS_A_BED_TC  "TC-7" %
%   N7:81  TC_OPEN_SP  "CONFIG The value read by an open TC input" %
%   N16:21  ADS_A_BED_TEMP_READ %
% Rung: 6 %
SOR NEQ I:5.6 N7:81 MOV I:5.6 N16:21 EOR
%   I:5.6  ADS_A_BED_TC  "TC-7" %
%   N7:81  TC_OPEN_SP  "CONFIG The value read by an open TC input" %
%   N16:21  ADS_A_BED_TEMP_READ %

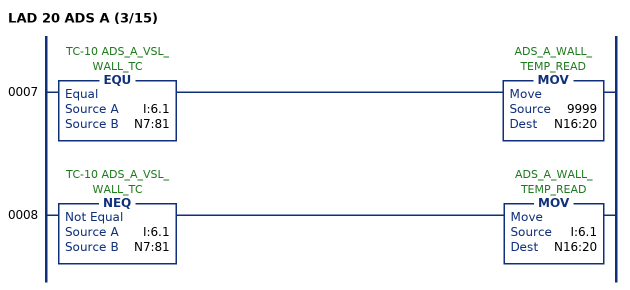
% Rung: 7 %
SOR EQU I:6.1 N7:81 MOV 9999 N16:20 EOR
%   I:6.1  ADS_A_VSL_WALL_TC  "TC-10" %
%   N7:81  TC_OPEN_SP  "CONFIG The value read by an open TC input" %
%   N16:20  ADS_A_WALL_TEMP_READ %
% Rung: 8 %
SOR NEQ I:6.1 N7:81 MOV I:6.1 N16:20 EOR
%   I:6.1  ADS_A_VSL_WALL_TC  "TC-10" %
%   N7:81  TC_OPEN_SP  "CONFIG The value read by an open TC input" %
%   N16:20  ADS_A_WALL_TEMP_READ %

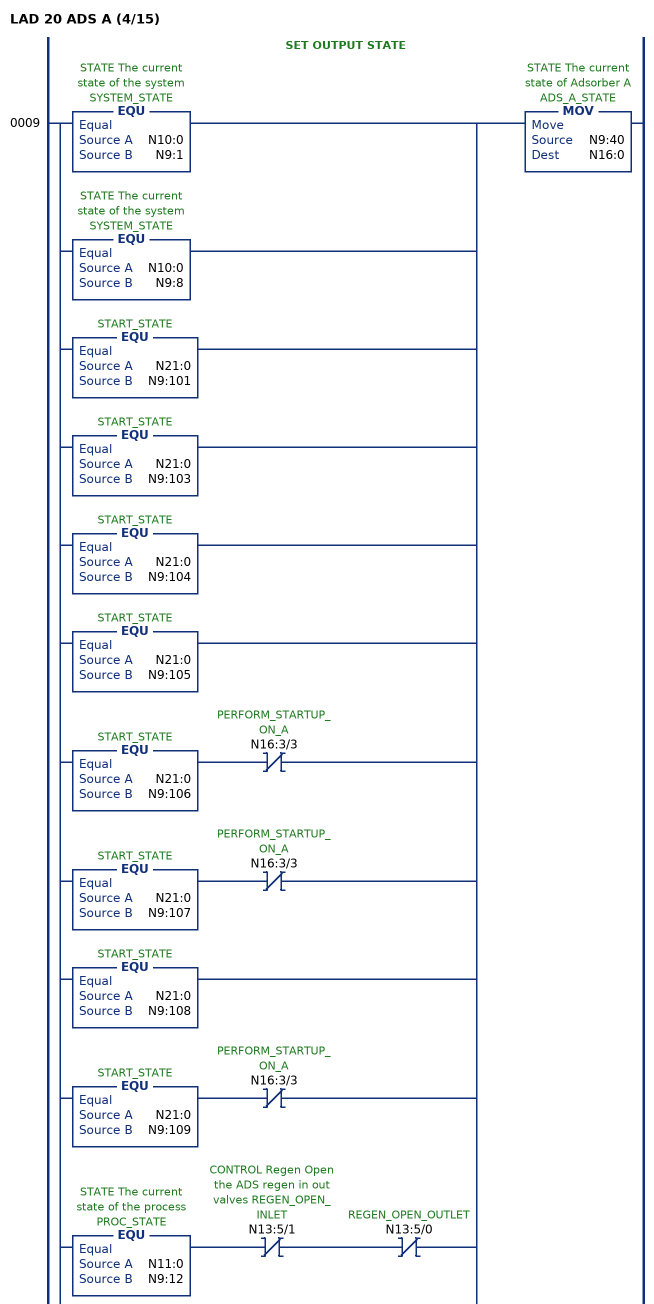

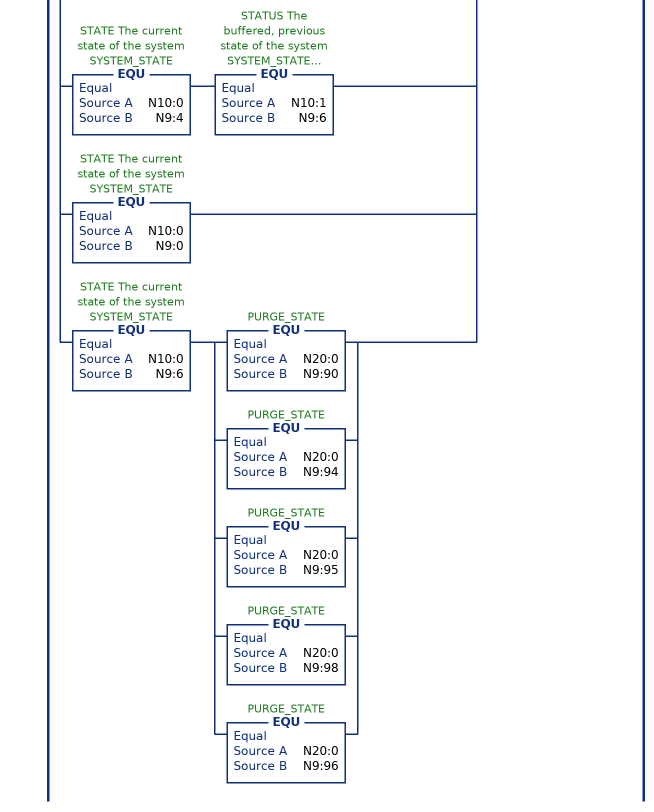
% Rung: 9 %
% TITLE: SET OUTPUT STATE %
SOR BST EQU N10:0 N9:1 NXB EQU N10:0 N9:8 NXB BST EQU N21:0 N9:101 NXB EQU N21:0 N9:103 NXB EQU N21:0 N9:104 NXB EQU N21:0 N9:105 NXB EQU N21:0 N9:106 XIO N16:3/3 NXB EQU N21:0 N9:107 XIO N16:3/3 NXB EQU N21:0 N9:108 NXB EQU N21:0 N9:109 XIO N16:3/3 BND NXB EQU N11:0 N9:12 XIO N13:5/1 XIO N13:5/0 NXB EQU N10:0 N9:4 EQU N10:1 N9:6 NXB EQU N10:0 N9:0 NXB EQU N10:0 N9:6 BST EQU N20:0 N9:90 NXB EQU N20:0 N9:94 NXB EQU N20:0 N9:95 NXB EQU N20:0 N9:98 NXB EQU N20:0 N9:96 BND BND MOV N9:40 N16:0 EOR
%   N10:0  SYSTEM_STATE  "STATE The current state of the system" %
%   N9:1  SYSTEM_STANDBY  "STATE System Process" %
%   N9:8  SYSTEM_SUPPLEMENTAL %
%   N21:0  START_STATE %
%   N9:101  START_COOL %
%   N9:103  START_VENT_GET_1 %
%   N9:104  START_HEAT_GETTER %
%   N9:105  START_VENT_ALL %
%   N9:106  START_BACKFILL_1 %
%   N16:3/3  PERFORM_STARTUP_ON_A %
%   N9:107  START_VENT_ADS_2 %
%   N9:108  START_VENT_GET_2 %
%   N9:109  START_BKFL_2 %
%   N11:0  PROC_STATE  "STATE The current state of the process" %
%   N9:12  PROC_PFY_B_REG_A  "STATE Process Purify B" %
%   N13:5/1  REGEN_OPEN_INLET  "CONTROL Regen Open the ADS regen in out valves" %
%   N13:5/0  REGEN_OPEN_OUTLET %
%   N9:4  SYSTEM_ALARM  "STATE System Alarm" %
%   N10:1  SYSTEM_STATE_BUFFER  "STATUS The buffered, previous state of the system" %
%   N9:6  SYSTEM_PURGE %
%   N9:0  SYSTEM_OFFLINE %
%   N20:0  PURGE_STATE %
%   N9:90  PURGE_IDLE %
%   N9:94  PURGE_FINAL_VENT %
%   N9:95  PURGE_DONE %
%   N9:98  PURGE_VENT_GET_2 %
%   N9:96  PURGE_VENT_GETTER %
%   N9:40  ADS_STANDBY  "STATE ADS Standby" %
%   N16:0  ADS_A_STATE  "STATE The current state of Adsorber A" %

